FUNCTION_BLOCK ABSTRACT CommunicatorSFC EXTENDS TC.ToolkitObject

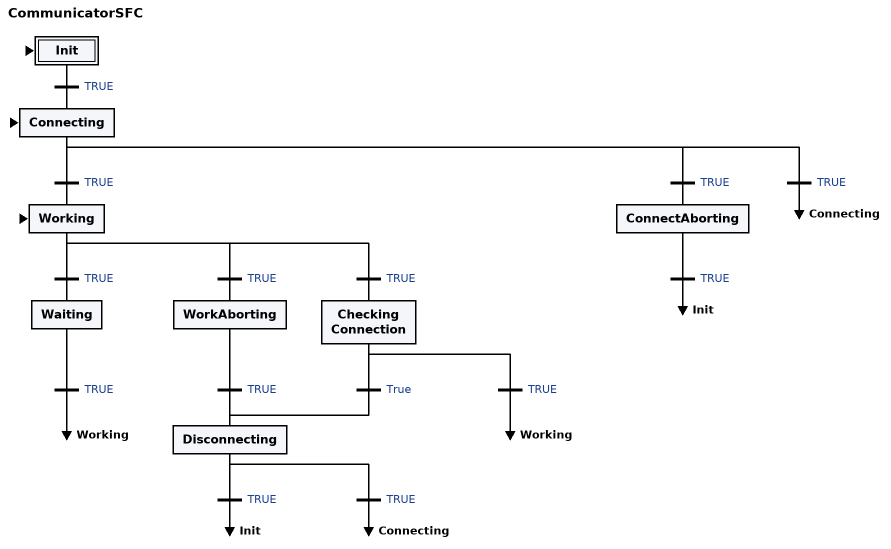
INITIAL_STEP Init:
END_STEP
TRANSITION FROM Init TO Connecting
    := TRUE;
END_TRANSITION
STEP Connecting:
END_STEP
TRANSITION FROM Connecting TO Working
    := TRUE;
END_TRANSITION
STEP Working:
END_STEP
TRANSITION FROM Connecting TO ConnectAborting
    := TRUE;
END_TRANSITION
STEP ConnectAborting:
END_STEP
TRANSITION FROM ConnectAborting TO Init
    := TRUE;
END_TRANSITION
TRANSITION FROM Connecting TO Connecting
    := TRUE;
END_TRANSITION
TRANSITION FROM Working TO Waiting
    := TRUE;
END_TRANSITION
STEP Waiting:
END_STEP
TRANSITION FROM Waiting TO Working
    := TRUE;
END_TRANSITION
TRANSITION FROM Working TO WorkAborting
    := TRUE;
END_TRANSITION
STEP WorkAborting:
END_STEP
TRANSITION FROM WorkAborting TO Disconnecting
    := TRUE;
END_TRANSITION
TRANSITION FROM Working TO CheckingConnection
    := TRUE;
END_TRANSITION
STEP CheckingConnection:
END_STEP
TRANSITION FROM CheckingConnection TO Disconnecting
    := True;
END_TRANSITION
TRANSITION FROM CheckingConnection TO Working
    := TRUE;
END_TRANSITION
STEP Disconnecting:
END_STEP
TRANSITION FROM Disconnecting TO Init
    := TRUE;
END_TRANSITION
TRANSITION FROM Disconnecting TO Connecting
    := TRUE;
END_TRANSITION

END_FUNCTION_BLOCK

(* stored: Version 1.1.0.1
   POU CommunicatorSFC: Id {bc996d58-2ab1-01ba-0c6e-599e3d7035da}, SpecialFunc None
   Folder Actions: Id {51586432-debb-05fc-2c12-591d8e6c9c68}
   Folder Transitions: Id {75cf2bfc-f11f-01b0-06f7-bc08ca3fcae2} *)
